PROGRAM main
VAR_INPUT
	X0 : bool;
	X1 : bool;
	X2 : bool;
	X3 : bool;
	X4 : bool;
	X5 : bool;
END_VAR

VAR_OUTPUT
	Y0 : bool;
	Y1 : bool;
END_VAR

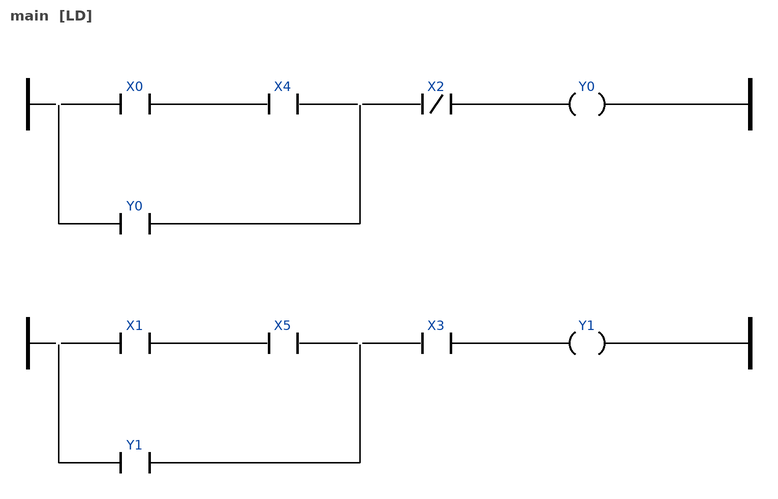
(* LD diagram, written out as Structured Text *)
Y0 := (Y0 OR X0 AND X4) AND NOT X2;
Y1 := (Y1 OR X1 AND X5) AND X3;
END_PROGRAM
